FUNCTION_BLOCK HandlingSequence EXTENDS ZApplication.Sequence
VAR
  {attribute 'hide'}
  _parent : REFERENCE TO HandlingUnit;
  _io : REFERENCE TO HandlingIo;
  _actuator : REFERENCE TO HandlingActuator;
  _fieldbus : REFERENCE TO HandlingFieldbus;
  _axis : REFERENCE TO HandlingAxis;
  _collision : REFERENCE TO HandlingCollision;  
  _data : REFERENCE TO HandlingDataRef;
  _unit : REFERENCE TO HandlingLinkedUnit;  
END_VAR

METHOD FB_init : BOOL
VAR_INPUT
  bInitRetains : BOOL; // if TRUE, the retain variables are initialized (warm start / cold start)
  bInCopyCode : BOOL;  // if TRUE, the instance afterwards gets moved into the copy code (online change)
  unit : REFERENCE TO HandlingUnit;
END_VAR
_parent REF= unit;
_alarming := unit._alarming;
_io REF= unit._equipment.Io;
_actuator REF= unit._equipment.Actuator;
_fieldbus REF= unit._equipment.Fieldbus;
_axis REF= unit._equipment.Axis;
_collision REF= unit._equipment.Collision;
_unit REF= unit._equipment.Unit;
_data REF= unit._data;
_loggerDiagnostics.SetLogger(unit._logger);
END_METHOD

METHOD StepDecoded : ZCore.ZString
VAR_INPUT
  stepIndex : INT;
END_VAR
VAR_INST
  _stepIndexDecoded : HandlingStep;
END_VAR
_stepIndexDecoded := stepIndex;
stepDecoded := TO_STRING(_stepIndexDecoded);
END_METHOD

END_FUNCTION_BLOCK

(* stored: Version 1.1.0.1
   POU HandlingSequence: Id {3346b6c8-767a-4fe9-8ab9-8756b683ca35}, SpecialFunc None
   Method FB_init: Id {989c67af-f97a-4d21-8ee5-cdf3e4da05e1}
   Method StepDecoded: Id {5231d17b-8eaf-4fc1-9952-77b1cbd1c31d} *)
